(* Logix 5000 project; controller jamiesFYP_PLC vendor 1 type 14 code 92 rev 35.12; software revision 35.01 *)

TASK MainTask (continuous, watchdog 500 ms) : MainProgram

MODULES
   Local : vendor 1 type 14 code 92 (ICP 0, rev 35.12)
      jamiesFYP_DCinput : vendor 1 type 7 code 2 (ICP 2, rev 3.1, Input RPI 20 ms)
      jamiesFYP_DCoutput : 1756-OB16D (ICP 1, rev 3.1, Output RPI 20 ms)
      jamiesFYP_Ethernet : 1756-EN2T (ICP 5, Ethernet 10.188.2.144, rev 11.1)
         GLW_LAB_LD_ROB01 : FANUC Robot R30iB Plus (Ethernet 10.188.2.186, rev 3.1, StandardDataDriven RPI 32 ms)
END_MODULES

VAR_GLOBAL   (* controller tags *)
   HMI_Start : BOOL;
   HMI_Stop : BOOL;
   LDRobot_AtFullView : ALIAS FOR GLW_LAB_LD_ROB01:I1.Input[3].3;   // Robot at Fluke Full View
   LDRobot_AtHomePos : ALIAS FOR GLW_LAB_LD_ROB01:I1.Input[3].0;   // Robot at Home Pos
   LDRobot_AtPos1 : ALIAS FOR GLW_LAB_LD_ROB01:I1.Input[3].1;   // Robot at Fluke Pos 1
   LDRobot_AtPos2 : ALIAS FOR GLW_LAB_LD_ROB01:I1.Input[3].2;   // Robot at Fluke Pos 2
   LDRobot_CycleComplete : ALIAS FOR GLW_LAB_LD_ROB01:I1.Input[3].4;   // Robot Cycle Complete
   LDRobot_CycleStop : ALIAS FOR GLW_LAB_LD_ROB01:O1.Output[0].3;
   LDRobot_Enable : ALIAS FOR GLW_LAB_LD_ROB01:O1.Output[0].7;
   LDRobot_FaultReset : ALIAS FOR GLW_LAB_LD_ROB01:O1.Output[0].4;
   LDRobot_Hold : ALIAS FOR GLW_LAB_LD_ROB01:O1.Output[0].1;
   LDRobot_IMSTP : ALIAS FOR GLW_LAB_LD_ROB01:O1.Output[0].0;
   LDRobot_SFSPD : ALIAS FOR GLW_LAB_LD_ROB01:O1.Output[0].2;
   LDRobot_Start : ALIAS FOR GLW_LAB_LD_ROB01:O1.Output[0].5;
END_VAR

PROGRAM MainProgram   (* main routine MainRoutine *)

ROUTINE MainRoutine   (* ladder *)
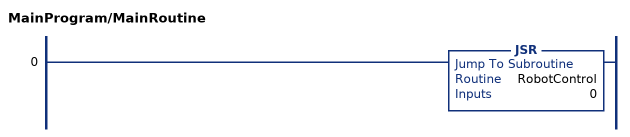
   0: JSR(RobotControl,0);
END_ROUTINE

ROUTINE RobotControl   (* ladder *)
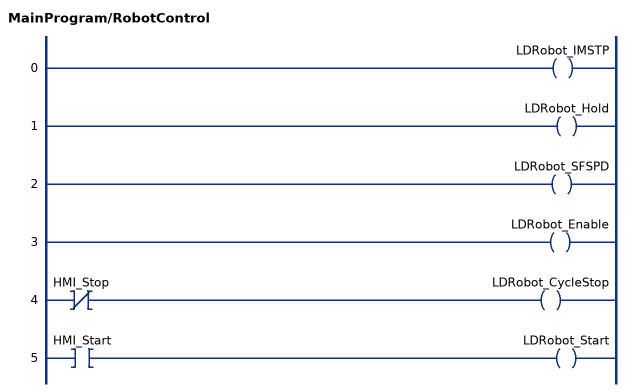
   0: OTE(LDRobot_IMSTP);
   1: OTE(LDRobot_Hold);
   2: OTE(LDRobot_SFSPD);
   3: OTE(LDRobot_Enable);
   4: XIO(HMI_Stop)OTE(LDRobot_CycleStop);
   5: XIC(HMI_Start)OTE(LDRobot_Start);
END_ROUTINE
END_PROGRAM
